FUNCTION_BLOCK OUT_ANY_CONSOLE (* Service Interface Function Block Type for debugging, tracing, etc. *)
  (* Description: Copyright (c) 2011 Profactor GmbH This program and the accompanying materials are made available under the terms of the Eclipse Public License 2.0 which is available at https://www.eclipse.org/legal/epl-2.0/ SPDX-License-Identifier: EPL-2.0 *)
  (* Version 1.0, 2011-08-29, Thomas Strasser, Profactor GmbH *)
  (* Version 3.0, 2025-04-14, Patrick Aigner, changed package *)
  PACKAGE eclipse4diac::utils;
  (* Compiler Cpp Unknown Unknown 1.0 *)
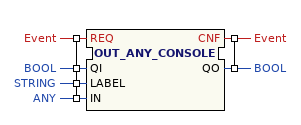
  EVENT_INPUT
    REQ WITH QI, IN, LABEL; (* Service Request *)
  END_EVENT
  EVENT_OUTPUT
    CNF WITH QO; (* Confirmation of Requested Service *)
  END_EVENT
  VAR_INPUT
    QI : BOOL; (* Event Input Qualifier *)
    LABEL : STRING; (* Label for the output value *)
    IN : ANY; (* Output value to console *)
  END_VAR
  VAR_OUTPUT
    QO : BOOL; (* Event Output Qualifier *)
  END_VAR
END_FUNCTION_BLOCK
